{attribute 'qualified_only'}
VAR_GLOBAL
 	/// 計測データ
	MeasuredData : ARRAY[1..10] OF LREAL;
END_VAR

(* stored: Version 1.1.0.1
   GVL GVL: Id {cb1bf10f-c647-4024-83a0-f157b155c910} *)
